Staubli VAL3: Path.pjx

--- Path.pjx ---
Parameters version=s7.8.3 stackSize=5000 millimeterUnit=true
Program file=Delete.pgx
Program file=EditMain.pgx
Program file=EditPathIn.pgx
Program file=EditPoint.pgx
Program file=EnterPageKey.pgx
Program file=getPtPara.pgx
Program file=Init.pgx
Program file=loadPath.pgx
Program file=Main.pgx
Program file=MainKey.pgx
Program file=OnF1.pgx
Program file=OnF2.pgx
Program file=OnF3.pgx
Program file=OnF4.pgx
Program file=OnF5.pgx
Program file=OnF6.pgx
Program file=OnF7.pgx
Program file=OnF8.pgx
Program file=readFileList.pgx
Program file=Refresh.pgx
Program file=Refresh1.pgx
Program file=Refresh2.pgx
Program file=Refresh3.pgx
Program file=RefreshList.pgx
Program file=Save.pgx
Program file=selectFile.pgx
Program file=setPara.pgx
Program file=SimuMain.pgx
Program file=start.pgx
Program file=stop.pgx
Data file=Path.dtx
Library alias=master path=Disk://template/normal/normal.pjx
Library alias=user path=Disk://userPage/USERPAGE.pjx
Library alias=PublicData path=Disk://PublicData/PublicData.pjx
Library alias=Tool path=Disk://Tool/Tool.pjx
Library alias=Frame path=Disk://Frame/Frame.pjx
Library alias=PublicProg path=Disk://PublicProg/PublicProg.pjx
Library alias=IO path=Disk://IO/IO.pjx
Library alias=SparePoint path=Disk://SparePoint/SparePoint.pjx
Library alias=Motion path=Disk://Motion/Motion.pjx
Library alias=prd path=Disk://template/normalPath/normalPath.pjx

--- Path.dtx ---
bool bByPass[4]
bool bExit
bool bListRefresh
bool bUserRefresh
mdesc mNomSpeed
num nPage = 1
num nSelected
public string sDeli[2]
  [0] = "A"
  [1] = "C"
public string sFileList = "A140"
string sFolder = "Disk://Traj/"
string sItem = "p1"
string sList[316]
  [0] = "p1"
  [1] = "p2"
  [2] = "p3"
  [3] = "p4"
  [4] = "p5"
  [5] = "p6"
  [6] = "p7"
  [7] = "p8"
  [8] = "p9"
  [9] = "p10"
  [10] = "p11"
  [11] = "p12"
  [12] = "p13"
  [13] = "p14"
  [14] = "p15"
  [15] = "p16"
  [16] = "p17"
  [17] = "p18"
  [18] = "p19"
  [19] = "p20"
  [20] = "p21"
  [21] = "p22"
  [22] = "p23"
  [23] = "p24"
  [24] = "p25"
  [25] = "p26"
  [26] = "p27"
  [27] = "p28"
  [28] = "p29"
  [29] = "p30"
  [30] = "p31"
  [31] = "p32"
  [32] = "p33"
  [33] = "p34"
  [34] = "p35"
  [35] = "p36"
  [36] = "p37"
  [37] = "p38"
  [38] = "p39"
  [39] = "p40"
  [40] = "p41"
  [41] = "p42"
  [42] = "p43"
  [43] = "p44"
  [44] = "p45"
  [45] = "p46"
  [46] = "p47"
  [47] = "p48"
  [48] = "p49"
  [49] = "p50"
  [50] = "p51"
  [51] = "p52"
  [52] = "p53"
  [53] = "p54"
  [54] = "p55"
  [55] = "p56"
  [56] = "p57"
  [57] = "p58"
  [58] = "p59"
  [59] = "p60"
  [60] = "p61"
  [61] = "p62"
  [62] = "p63"
  [63] = "p64"
  [64] = "p65"
  [65] = "p66"
  [66] = "p67"
  [67] = "p68"
  [68] = "p69"
  [69] = "p70"
  [70] = "p71"
  [71] = "p72"
  [72] = "p73"
  [73] = "p74"
  [74] = "p75"
  [75] = "p76"
  [76] = "p77"
  [77] = "p78"
  [78] = "p79"
  [79] = "p80"
  [80] = "p81"
  [81] = "p82"
  [82] = "p83"
  [83] = "p84"
  [84] = "p85"
  [85] = "p86"
  [86] = "p87"
  [87] = "p88"
  [88] = "p89"
  [89] = "p90"
  [90] = "p91"
  [91] = "p92"
  [92] = "p93"
  [93] = "p94"
  [94] = "p95"
  [95] = "p96"
  [96] = "p97"
  [97] = "p98"
  [98] = "p99"
  [99] = "p100"
  [100] = "p101"
  [101] = "p102"
  [102] = "p103"
  [103] = "p104"
  [104] = "p105"
  [105] = "p106"
  [106] = "p107"
  [107] = "p108"
  [108] = "p109"
  [109] = "p110"
  [110] = "p111"
  [111] = "p112"
  [112] = "p113"
  [113] = "p114"
  [114] = "p115"
  [115] = "p116"
  [116] = "p117"
  [117] = "p118"
  [118] = "p119"
  [119] = "p120"
  [120] = "p121"
  [121] = "p122"
  [122] = "p123"
  [123] = "p124"
  [124] = "p125"
  [125] = "p126"
  [126] = "p127"
  [127] = "p128"
  [128] = "p129"
  [129] = "p130"
  [130] = "p131"
  [131] = "p132"
  [132] = "p133"
  [133] = "p134"
  [134] = "p135"
  [135] = "p136"
  [136] = "p137"
  [137] = "p138"
  [138] = "p139"
  [139] = "p140"
  [140] = "p141"
  [141] = "p142"
  [142] = "p143"
  [143] = "p144"
  [144] = "p145"
  [145] = "p146"
  [146] = "p147"
  [147] = "p148"
  [148] = "p149"
  [149] = "p150"
  [150] = "p151"
  [151] = "p152"
  [152] = "p153"
  [153] = "p154"
  [154] = "p155"
  [155] = "p156"
  [156] = "p157"
  [157] = "p158"
  [158] = "p159"
  [159] = "p160"
  [160] = "p161"
  [161] = "p162"
  [162] = "p163"
  [163] = "p164"
  [164] = "p165"
  [165] = "p166"
  [166] = "p167"
  [167] = "p168"
  [168] = "p169"
  [169] = "p170"
  [170] = "p171"
  [171] = "p172"
  [172] = "p173"
  [173] = "p174"
  [174] = "p175"
  [175] = "p176"
  [176] = "p177"
  [177] = "p178"
  [178] = "p179"
  [179] = "p180"
  [180] = "p181"
  [181] = "p182"
  [182] = "p183"
  [183] = "p184"
  [184] = "p185"
  [185] = "p186"
  [186] = "p187"
  [187] = "p188"
  [188] = "p189"
  [189] = "p190"
  [190] = "p191"
  [191] = "p192"
  [192] = "p193"
  [193] = "p194"
  [194] = "p195"
  [195] = "p196"
  [196] = "p197"
  [197] = "p198"
  [198] = "p199"
  [199] = "p200"
  [200] = "p201"
  [201] = "p202"
  [202] = "p203"
  [203] = "p204"
  [204] = "p205"
  [205] = "p206"
  [206] = "p207"
  [207] = "p208"
  [208] = "p209"
  [209] = "p210"
  [210] = "p211"
  [211] = "p212"
  [212] = "p213"
  [213] = "p214"
  [214] = "p215"
  [215] = "p216"
  [216] = "p217"
  [217] = "p218"
  [218] = "p219"
  [219] = "p220"
  [220] = "p221"
  [221] = "p222"
  [222] = "p223"
  [223] = "p224"
  [224] = "p225"
  [225] = "p226"
  [226] = "p227"
  [227] = "p228"
  [228] = "p229"
  [229] = "p230"
  [230] = "p231"
  [231] = "p232"
  [232] = "p233"
  [233] = "p234"
  [234] = "p235"
  [235] = "p236"
  [236] = "p237"
  [237] = "p238"
  [238] = "p239"
  [239] = "p240"
  [240] = "p241"
  [241] = "p242"
  [242] = "p243"
  [243] = "p244"
  [244] = "p245"
  [245] = "p246"
  [246] = "p247"
  [247] = "p248"
  [248] = "p249"
  [249] = "p250"
  [250] = "p251"
  [251] = "p252"
  [252] = "p253"
  [253] = "p254"
  [254] = "p255"
  [255] = "p256"
  [256] = "p257"
  [257] = "p258"
  [258] = "p259"
  [259] = "p260"
  [260] = "p261"
  [261] = "p262"
  [262] = "p263"
  [263] = "p264"
  [264] = "p265"
  [265] = "p266"
  [266] = "p267"
  [267] = "p268"
  [268] = "p269"
  [269] = "p270"
  [270] = "p271"
  [271] = "p272"
  [272] = "p273"
  [273] = "p274"
  [274] = "p275"
  [275] = "p276"
  [276] = "p277"
  [277] = "p278"
  [278] = "p279"
  [279] = "p280"
  [280] = "p281"
  [281] = "p282"
  [282] = "p283"
  [283] = "p284"
  [284] = "p285"
  [285] = "p286"
  [286] = "p287"
  [287] = "p288"
  [288] = "p289"
  [289] = "p290"
  [290] = "p291"
  [291] = "p292"
  [292] = "p293"
  [293] = "p294"
  [294] = "p295"
  [295] = "p296"
  [296] = "p297"
  [297] = "p298"
  [298] = "p299"
  [299] = "p300"
  [300] = "p301"
  [301] = "p302"
  [302] = "p303"
  [303] = "p304"
  [304] = "p305"
  [305] = "p306"
  [306] = "p307"
  [307] = "p308"
  [308] = "p309"
  [309] = "p310"
  [310] = "p311"
  [311] = "p312"
  [312] = "p313"
  [313] = "p314"
  [314] = "p315"
  [315] = "p316"
string sListItemValue
string sOutputFolder = "Disk://Traj/"
string sParameter
string sPtPara
frame fFrame = {fatherId=world[0]}
tool tTool = {fatherId=flange[0], ioLink=valve1}
pointRx pTemp = {fatherId=world[0]}

--- start.pgx ---
public program start()
begin
  //
  call Init()
  call Main()
end

--- Delete.pgx ---
program Delete()
  local string l_sYesNo[2]
  local num l_i
begin
  //删除
  l_sYesNo[0]="是"
  l_sYesNo[1]="否"
  switch nPage
    case 0
      call user:questionDialog("是否删除此路径?",l_sYesNo,l_i)
      if l_i==0 or l_i==1
        if size(sFileList)==1
          if sFileList[nSelected]!=""
            libDelete(sFolder+sFileList[nSelected])
            sFileList[nSelected]=""
            bListRefresh=true
          endIf
        else
          libDelete(sFolder+sFileList[nSelected])
          delete(sFileList[nSelected])
          bListRefresh=true
        endIf

      endIf
    break
    case 1
      call user:questionDialog("是否删除此点?",l_sYesNo,l_i)
      if l_i==0 or l_i==1
        if sFileList[nSelected]!=""
          delete(prd:pDemo[nSelected])
          delete(prd:sPtParameter[nSelected])
          bListRefresh=true
        endIf
      endIf
    break
  endSwitch

  bUserRefresh=true
end

--- EditPathIn.pgx ---
public program EditPathIn(string x_sPath)
  local num l_nKey
  local bool l_bRes
begin
  //

  //
  //load path

    call loadPath(l_bRes,x_sPath)
    if !l_bRes
      return
    endIf

    //
    bUserRefresh=bListRefresh=true
    nPage=1
    //
    do
      call Refresh1()
      call RefreshList()
      call user:setList(x_sPath,sList,bUserRefresh,bListRefresh,nSelected,sItem,l_nKey)
      bUserRefresh=false
      bListRefresh=false
      call MainKey(l_nKey)
      delay(0)
    until bExit
    nPage=0
    bExit=false
    bUserRefresh=bListRefresh=true

end

--- EditPoint.pgx ---
program EditPoint()
  local bool l_bRes
  local num l_i
  local string l_sValue
  local num l_nSelect
  local string l_sItem
  local num l_nKey
  local num l_nRes
begin
  switch nPage
    //运动点
    case 1
      cls()
      resize(sParameter,1,12)
      sParameter[0]="X"
      sParameter[1]="Y"
      sParameter[2]="Z"
      sParameter[3]="Rx"
      sParameter[4]="Ry"
      sParameter[5]="Rz"
      sParameter[6]="PIn1"
      sParameter[7]="PIn2"
      sParameter[8]="POut"
      sParameter[9]="IO1"
      sParameter[10]="IO2"
      sParameter[11]="delay"
      //
      resize(sListItemValue,1,size(sParameter))
      sListItemValue[0]=toString(".3",prd:pDemo[nSelected].trsf.x)
      sListItemValue[1]=toString(".3",prd:pDemo[nSelected].trsf.y)
      sListItemValue[2]=toString(".3",prd:pDemo[nSelected].trsf.z)
      sListItemValue[3]=toString(".3",prd:pDemo[nSelected].trsf.rx)
      sListItemValue[4]=toString(".3",prd:pDemo[nSelected].trsf.ry)
      sListItemValue[5]=toString(".3",prd:pDemo[nSelected].trsf.rz)
      //解析sPtParameter
      call getPtPara(prd:sPtParameter[nSelected],sPtPara)
      sListItemValue[6]=sPtPara[0]
      sListItemValue[7]=sPtPara[1]
      sListItemValue[8]=sPtPara[2]
      sListItemValue[9]=sPtPara[3]
      sListItemValue[10]=sPtPara[4]
      sListItemValue[11]=sPtPara[5]
      //
      for l_i=0 to size(sParameter)-1
        call user:strlength(sParameter[l_i],user:nBottomX/2)
        l_sValue=sListItemValue[l_i]
        call user:strlength(l_sValue,user:nBottomX/2+1)
        sParameter[l_i]=sParameter[l_i]+":"+l_sValue
      endFor

      bUserRefresh=true
      bListRefresh=true
      //
      do
        if bUserRefresh
          cls()
          call user:clear(0,13)
          call user:typeMenu(8,"确定")
        endIf
        call user:setList("编辑点",sParameter,bUserRefresh,bListRefresh,l_nSelect,l_sItem,l_nKey)
        bUserRefresh=false
        bListRefresh=false
        call EnterPageKey(l_nKey,l_nSelect,sParameter[l_nSelect])
        delay(0)
      until l_nKey==255 or l_nKey==278
      prd:sPtParameter[nSelected]=sListItemValue[6]+"/"+sListItemValue[7]+"/"+sListItemValue[8]+"/"+sListItemValue[9]+"/"+sListItemValue[10]+"/"+sListItemValue[11]
      bUserRefresh=true
      bListRefresh=true
    break
  endSwitch
end

--- EnterPageKey.pgx ---
program EnterPageKey(num& x_nKey, num& x_nSelect, string& x_sItem)
  local string l_sStr
  local num l_nKey
  local string l_sEmpty
  local string l_sValue
  local num l_nItem
  local num l_nView
  local string l_sItem
  local point lp
  local string l_sYN[2]
  local bool l_bRes
  local num l_nTemp
begin
  //
  //编辑项目
  switch x_nSelect
    //X
    case 0
      if x_nKey==270
        call user:editNum(x_sItem,sListItemValue[x_nSelect],prd:pDemo[nSelected].trsf.x,x_nSelect)
      endIf
    break
    //Y
    case 1
      if x_nKey==270
        call user:editNum(x_sItem,sListItemValue[x_nSelect],prd:pDemo[nSelected].trsf.y,x_nSelect)
      endIf
    break
    //Z
    case 2
      if x_nKey==270
        call user:editNum(x_sItem,sListItemValue[x_nSelect],prd:pDemo[nSelected].trsf.z,x_nSelect)
      endIf
    break
    //rx
    case 3
      if x_nKey==270
        call user:editNum(x_sItem,sListItemValue[x_nSelect],prd:pDemo[nSelected].trsf.rx,x_nSelect)
      endIf
    break
    //ry
    case 4
      if x_nKey==270
        call user:editNum(x_sItem,sListItemValue[x_nSelect],prd:pDemo[nSelected].trsf.ry,x_nSelect)
      endIf
    break
    //rz
    case 5
      if x_nKey==270
        call user:editNum(x_sItem,sListItemValue[x_nSelect],prd:pDemo[nSelected].trsf.rz,x_nSelect)
      endIf
    break
    //PIn1
    case 6
      if x_nKey==270
        call SparePoint:setPoint(sListItemValue[x_nSelect])
        call SparePoint:start()
        call SparePoint:getPoint(sListItemValue[x_nSelect])
        x_sItem="PIn1     :"+sListItemValue[x_nSelect]
      endIf

    break
    //PIn2
    case 7
      if x_nKey==270
        call SparePoint:setPoint(sListItemValue[x_nSelect])
        call SparePoint:start()
        call SparePoint:getPoint(sListItemValue[x_nSelect])
        x_sItem="PIn2     :"+sListItemValue[x_nSelect]
      endIf
    break
    //POut1
    case 8
      if x_nKey==270
        call SparePoint:setPoint(sListItemValue[x_nSelect])
        call SparePoint:start()
        call SparePoint:getPoint(sListItemValue[x_nSelect])
        x_sItem="POut     :"+sListItemValue[x_nSelect]
      endIf
    break
    //IO1
    case 9
      if x_nKey==270
        call IO:setIO(sListItemValue[x_nSelect])
        call IO:Main(1)
        call IO:getIO(sListItemValue[x_nSelect])
        //
        x_sItem="IO1      :"+sListItemValue[x_nSelect]
      endIf

    break
    //IO2
    case 10
      if x_nKey==270
        call IO:setIO(sListItemValue[x_nSelect])
        call IO:Main(1)
        call IO:getIO(sListItemValue[x_nSelect])
        //
        x_sItem="IO2      :"+sListItemValue[x_nSelect]
      endIf
    break
    //delay
    case 11
      if x_nKey==270
        call user:editNum(x_sItem,sListItemValue[x_nSelect],l_nTemp,x_nSelect)
      endIf
    break
  endSwitch
  if x_nKey==270
    bUserRefresh=true
    bListRefresh=true
  endIf
end

--- getPtPara.pgx ---
program getPtPara(string x_sPtPara, string& x_sOutPtpara[])
  local num l_nRes
  local num l_ni
begin
  //对参数x_sPtPara进行解析，得到相应信息
  //x_sPtPara结构：p1/p2/IO1/IO2/0.1
  //若没有，使用-1代替
  call PublicProg:SplitChar(l_nRes,x_sPtPara,"/",x_sOutPtpara)

end

--- Init.pgx ---
program Init()
  local num l_ni
begin
  //
  bUserRefresh=bListRefresh=true
  //
  bExit=false
  //
  call readFileList(sFolder,sFileList)
  //call selectFile(sDeli,sFileList)
  //

end

--- MainKey.pgx ---
program MainKey(num x_nKey)
  local num l_nKey
begin
  //
  switch x_nKey
    //编辑
    case 271
      call OnF1()
    break
    //取反
    case 272
      call OnF2()
    break
    //删除
    case 273
      call OnF3()
    break
    //工具、坐标系
    case 274
      call OnF4()
    break
    //
    case 275
    break
    //
    case 276
      call OnF6()
    break
    //save
    case 277
      call OnF7()
    break
    //返回
    case 278,255
      call OnF8("是否返回")
    break
    case 270
      call EditPoint()
    break
  endSwitch
  wait(getKey()==-1)
end

--- OnF1.pgx ---
program OnF1()
  local bool l_bRes
begin

  switch nPage
    case 0
      //编辑路径
      call EditMain(sItem)
    break
    case 1
      //
      tTool.trsf=Tool:tTool[prd:sToolName].trsf
      fFrame.trsf=Frame:fFrame[prd:sFrameName].trsf
      pTemp=here(tTool,fFrame)
      prd:pDemo[nSelected].trsf=pTemp.trsf
    break
    case 2
      //开始


    break
    case 3
    break
    case 4
    break

  endSwitch
end

--- OnF2.pgx ---
program OnF2()
  local num l_ni
  local bool l_bRes
begin
  switch nPage
    case 0
      //模拟
      call Motion:SimuMain(sItem)
      bUserRefresh=bListRefresh=true
    break
    case 1
      //insert
      nSelected=nSelected+1
      insert(prd:pDemo[nSelected])
      prd:pDemo[nSelected]=here(Tool:tTool[prd:sToolName],Frame:fFrame[prd:sFrameName])
      insert(prd:sPtParameter[nSelected])
      //添加点的信息
    break
    case 2
      //停止运动
    break
    case 3
    break
    case 4
    break

  endSwitch

end

--- OnF4.pgx ---
program OnF4()
  local string l_sProperty[2]
  local string l_sItem
begin
  //调用tool or frame library
  l_sProperty[0]="工具"
  l_sProperty[1]="坐标系"
  call user:SetProerty("",26,9,6,2,l_sProperty,l_sItem)
  if l_sItem=="工具"
    call Tool:setTool(prd:sToolName)
    call Tool:Main(1)
    call Tool:getTool(prd:sToolName,prd:tTool)
  elseIf l_sItem=="坐标系"
    call Frame:SetFrame(prd:sFrameName)
    call Frame:Main(1)
    call Frame:getFrame(prd:sFrameName,prd:fFrmMaster)
  endIf
  bUserRefresh=bListRefresh=true
end

--- OnF6.pgx ---
program OnF6()
  local string l_sTemp
begin
  //参数
  call setPara()
end

--- Refresh.pgx ---
program Refresh()
begin
  //
  if bUserRefresh
    cls()
    userPage()
    gotoxy(1,1)
    put("F1->编辑")
    gotoxy(1,13)
    put("F1")
    gotoxy(1,2)
    put("F2->模拟")
    gotoxy(6,13)
    put("F2")
    gotoxy(1,3)
    put("F3->删除")
    gotoxy(11,13)
    put("F3")
//    gotoxy(1,4)
//    put("F4->编辑路径")
//    gotoxy(16,13)
//    put("编辑")
    //
//    gotoxy(1,6)
//    put("F6->")
//    gotoxy(26,13)
//    put("")
//    gotoxy(1,7)
//    put("F7->")
//    gotoxy(31,13)
//    put("")
    gotoxy(1,7)
    put("F8->返回")
    gotoxy(36,13)
    put("F8")
  endIf
end

--- Refresh1.pgx ---
program Refresh1()
begin
  //编辑界面
  if bUserRefresh
    cls()
    userPage()
    gotoxy(1,1)
    put("F1->记录")
    gotoxy(1,13)
    put("F1")
    gotoxy(1,2)
    put("F2->插入")
    gotoxy(6,13)
    put("F2")
    gotoxy(1,3)
    put("F3->删除")
    gotoxy(11,13)
    put("F3")
    gotoxy(1,4)
    put("F4->选择工具/坐标系")
    gotoxy(16,13)
    put("F4")

    gotoxy(1,5)
    put("F5->运动方向切换")
    gotoxy(21,13)
    put("F5")
    gotoxy(1,6)
    put("F6->参数")
    gotoxy(26,13)
    put("F6")
    gotoxy(1,7)
    put("F7->保存")
    gotoxy(31,13)
    put("F7")
    gotoxy(1,8)
    put("F8->返回")
    gotoxy(36,13)
    put("F8")

    //
    gotoxy(1,10)
    put("工具："+prd:sToolName)
    gotoxy(1,11)
    put("坐标系："+prd:sFrameName)
  endIf
end

--- Refresh3.pgx ---
program Refresh3()
begin
  //选择工具/坐标系界面
  if bUserRefresh
    cls()
    userPage()
    gotoxy(1,1)
    put("F1->确定")
    gotoxy(1,13)
    put("F1")
    gotoxy(1,2)
    put("F2->编辑")
    gotoxy(6,13)
    put("F2")
//    gotoxy(1,3)
//    put("F3->删除")
//    gotoxy(11,13)
//    put("F3")
//    gotoxy(1,4)
//    put("F4->选择工具/坐标系")
//    gotoxy(16,13)
//    put("F4")
    //
//    gotoxy(1,6)
//    put("F6->")
//    gotoxy(26,13)
//    put("")
    gotoxy(1,7)
    put("F7->保存")
    gotoxy(31,13)
    put("F7")
    gotoxy(1,8)
    put("F8->返回")
    gotoxy(36,13)
    put("F8")
  endIf
end

--- RefreshList.pgx ---
program RefreshList()
  local num l_ni
begin
  //
  switch nPage
    //
    case 0
      if bListRefresh
        resize(sList,1,size(sFileList))
        for l_ni=0 to size(sFileList)-1
          sList[l_ni]=sFileList[l_ni]
        endFor
      endIf
    break
    //
    case 1
      if bListRefresh
        resize(sList,1,size(prd:pDemo))
        for l_ni=0 to size(prd:pDemo)-1
          sList[l_ni]="p"+toString("",l_ni+1)
        endFor
      endIf
    break
    case 2
    break
  endSwitch


end

--- Save.pgx ---
program Save()
  local num l_ni
begin
  //
  prd:libSave()
  popUpMsg("保存完毕!")
end

--- setPara.pgx ---
program setPara()
  local num l_nSelect
  local string l_sItem
  local num l_nKey
  local num l_i
  local string l_sValue
begin
  cls()
  resize(sParameter,1,3)
  sParameter[0]="补偿量"
  sParameter[1]="关节速度"
  sParameter[2]="直线速度"

  //
  resize(sListItemValue,1,size(sParameter))
  sListItemValue[0]=toString(".3",prd:nCompDelta)
  sListItemValue[1]=toString(".3",prd:mJoint.tvel)
  sListItemValue[2]=toString(".3",prd:mNormal.tvel)

  //
  for l_i=0 to size(sParameter)-1
    call user:strlength(sParameter[l_i],user:nBottomX/2)
    l_sValue=sListItemValue[l_i]
    call user:strlength(l_sValue,user:nBottomX/2+1)
    sParameter[l_i]=sParameter[l_i]+":"+l_sValue
  endFor

  bUserRefresh=true
  bListRefresh=true
  //
  do
    if bUserRefresh
      cls()
      call user:clear(0,13)
      call user:typeMenu(8,"确定")
    endIf
    call user:setList("参数",sParameter,bUserRefresh,bListRefresh,l_nSelect,l_sItem,l_nKey)
    bUserRefresh=false
    bListRefresh=false
    if l_nKey==270
      switch l_nSelect
        case 0
          call user:editNum(l_sItem,sListItemValue[l_nSelect],prd:nCompDelta,l_nSelect)
        break
        case 1
          call user:editNum(l_sItem,sListItemValue[l_nSelect],prd:mJoint.tvel,l_nSelect)
        break
        case 2
          call user:editNum(l_sItem,sListItemValue[l_nSelect],prd:mNormal.tvel,l_nSelect)
        break
      endSwitch
    endIf
      delay(0)
  until l_nKey==255 or l_nKey==278

  bUserRefresh=true
  bListRefresh=true
end
